PROGRAM TestToolkitBase
VAR
	testAutomationUnit : TestAutomationUnit;
	automationUnits : ARRAY [0..0] OF TwinCAT_OpenFramework_AutomationEngine.IAutomationUnit := [testAutomationUnit];
	
	automationEngine : TwinCAT_OpenFramework_AutomationEngine.AutomationEngine;
END_VAR

automationEngine.Run(automationUnits);

END_PROGRAM

(* stored: Version 1.1.0.1, ProductVersion 3.1.4026.12
   POU TestToolkitBase: Id {e4eb2eaa-3c4c-0200-2bd5-f94fd2ee20dd}, SpecialFunc None *)
